{attribute 'pack_mode' := '1'}
TYPE ST_CalibHeaderTest :
STRUCT
    sCalibrationNo : STRING(30);
    sUserId        : STRING(50);
END_STRUCT
END_TYPE

(* stored: Version 1.1.0.1, ProductVersion 3.1.4024.15
   DUT ST_CalibHeaderTest: Id {6dd872ba-10ca-4b13-bf37-fcef8bb2888a} *)
